{attribute addProperty BoxType "AX8206-0000-0041-0041"}
{attribute addProperty Id "Ch_B_Velocity_sensor_actual_value_invalidAT %I*BOOL811Ch_B_Position_actual_value_invalidAT %I*BOOL812Ch_B_1st_Additional_position_actual_value_invalidAT %I*BOOL813Ch_B_2nd_Additional_position_actual_value_invalidAT %I*BOOL814Ch_B_StatuswordAT %I*UINT1620Ch_B_Position_actual_valueAT %I*DINT3240Ch_B_Velocity_actual_valueAT %I*DINT3240"}
{attribute addProperty CRC "4097840841"}
{attribute addProperty SizeInBites "112"}
{attribute addProperty SizeInBytes "14"}
TYPE Ch_B_AxisMain_Inputs_F44016C9 :
STRUCT
	{attribute addProperty Name "Ch_B_Velocity_sensor_actual_value_invalid"}
	Ch_B_Velocity_sensor_actual_value_invalid AT %I* : BOOL;
	{attribute addProperty Name "Ch_B_Position_actual_value_invalid"}
	Ch_B_Position_actual_value_invalid AT %I* : BOOL;
	{attribute addProperty Name "Ch_B_1st_Additional_position_actual_value_invalid"}
	Ch_B_1st_Additional_position_actual_value_invalid AT %I* : BOOL;
	{attribute addProperty Name "Ch_B_2nd_Additional_position_actual_value_invalid"}
	Ch_B_2nd_Additional_position_actual_value_invalid AT %I* : BOOL;
	{attribute addProperty Name "Ch_B_Statusword"}
	Ch_B_Statusword AT %I* : UINT;
	{attribute addProperty Name "Ch_B_Position_actual_value"}
	Ch_B_Position_actual_value AT %I* : DINT;
	{attribute addProperty Name "Ch_B_Velocity_actual_value"}
	Ch_B_Velocity_actual_value AT %I* : DINT;
END_STRUCT
END_TYPE

(* stored: Version 1.2.0.0, ProductVersion 3.1.4024.9
   DUT Ch_B_AxisMain_Inputs_F44016C9: Id {e252e839-10c6-414a-a3fc-769899bbb85d} *)
